Fanuc KAREL source: ks00056.KL

-- PROVISIONAL review KL for V940-1; original PC SHA256 7f39cf4e09b1209ceb3c6f7597079831668b90c44e4a9673a4a11cfb63da514b
-- Incomplete behavior may be omitted. Consult companion uncertainty JSON. Do not deploy.
PROGRAM KS00056
%NOLOCKGROUP
BEGIN
  -- V9_ZERO_TABLE_METADATA_HINT layout=0001; no indexed target words; source/name/runtime held
  -- UNRESOLVED_PC offsets 5-13; opcodes 3F,75
  -- UNRESOLVED_PC offsets 18-27; opcodes 3F,75
  -- UNRESOLVED_PC offsets 32-70; opcodes 27,22,22,2A,22,2A,22,22,B0
  -- UNRESOLVED_PC offsets 75-79; opcodes 7F
END KS00056
